FUNCTION_BLOCK Test_F_UDINT_TO_DINT_Conversion EXTENDS T_UnitTestBase
VAR
    InputValue     : UDINT;
    ConvertedValue : DINT;
	Assertion : T_Assertion;
END_VAR

{attribute 'analysis' := '-33'} // inhibit unused variable warning
METHOD RunTest
VAR_OUTPUT
    TestCompleted : BOOL;
    TestFailed    : BOOL;
END_VAR
InputValue     := 2147483648;                  // too big
ConvertedValue := F_UDINT_TO_DINT(InputValue); // limit to largest DINT

TestFailed S= NOT Assertion.AssertEquals_DINT(Source    := TestName,
                             Expected     := 2147483647,
                            Actual       := ConvertedValue,
                            VariableName := 'ConvertedValue');

TestCompleted := TRUE;
END_METHOD

END_FUNCTION_BLOCK

(* stored: Version 1.1.0.1, ProductVersion 3.1.4024.12
   POU Test_F_UDINT_TO_DINT_Conversion: Id {0f7dcc90-c1e5-4697-8983-52848bcba636}, SpecialFunc None
   Method RunTest: Id {4aeb1853-9057-45ad-afb4-122c04cd546c} *)
